TYPE DUT_MODULE_INTERFACE_OUTPUT :
STRUCT
	///Free to use = TRUE, busy to use =FALSE
	Dummy: BOOL := TRUE;
	///Individual name of the module
	Name: STRING(80);
	///Identification number of module
	ID: UINT;
	///IP address
	IP: STRING(80);
	///Show if the module is in Standby or not
	Idle: BOOL;
	///Show if the module is connected
	Connected: BOOL;
	///Feedback with conection test input
	ConnectionTestOutput: BOOL;
	///Show if the system has error when=TRUE
	Error: BOOL;
	///Identification number of the error
	ErrorID: UINT;
	///Description of the error
	ErrorDescription: STRING(80);
	///Description of the current task
	CurrentTaskDescription: STRING(80);
	///actual position of the modules, calculated by the module itself
	PositionOutput: LREAL;
	///Position of the sensor
	PositionSensor: BOOL;
	///Range of OUTPUT skills
	SkillOutput: ARRAY[0..SkillCnt] OF DUT_SKILL_OUTPUT;
	///Range of state values
	StateValue: ARRAY[0..StateCnt] OF DUT_STATEVALUES;
END_STRUCT
END_TYPE

(* stored: Version 1.1.0.1, ProductVersion 3.1.0.25
   DUT DUT_MODULE_INTERFACE_OUTPUT: Id {465778e5-8710-4421-8d2f-57be97a5f311} *)
